TYPE ST_MCRelativeInput :
STRUCT
	Distance			:LREAL;
	Velocity  			:LREAL;
	Acceleration  		:LREAL;
	Deceleration 	 	:LREAL;
	Jerk				:LREAL;
	Execute  			:BOOL:=FALSE;
	boolbuf1			:BOOL;
	boolbuf2			:BOOL;
	boolbuf3			:BOOL;
	boolbuf4			:BOOL;
	boolbuf5			:BOOL;
	boolbuf6			:BOOL;
	boolbuf7			:BOOL;
END_STRUCT
END_TYPE

(* stored: Version 1.1.0.1, ProductVersion 3.1.4024.9
   DUT ST_MCRelativeInput: Id {581fa56b-b28e-4bbc-90f2-a0c247967fdd} *)
